FUNCTION_BLOCK PhysicsRulesWorkPieces (* Basic Function Block Type *)
  (* Standard: 61499-2 *)
  (* Version 0.0, 6/8/2016, Andrei, nxtControl GmbH, Template *)
  PACKAGE Main;
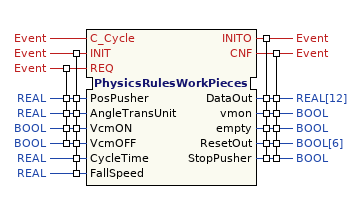
  EVENT_INPUT
    C_Cycle;
    INIT WITH PosPusher, AngleTransUnit, VcmON, VcmOFF, CycleTime, FallSpeed;
    REQ WITH PosPusher, AngleTransUnit, VcmON, VcmOFF; (* Normal Execution Request *)
  END_EVENT
  EVENT_OUTPUT
    INITO WITH DataOut, vmon, empty, ResetOut, StopPusher;
    CNF WITH DataOut, vmon, empty, ResetOut, StopPusher; (* Execution Confirmation *)
  END_EVENT
  VAR_INPUT
    PosPusher : REAL;
    AngleTransUnit : REAL;
    VcmON : BOOL;
    VcmOFF : BOOL;
    CycleTime : REAL;
    FallSpeed : REAL;
  END_VAR
  VAR_OUTPUT
    DataOut : ARRAY [0..11] OF REAL;
    vmon : BOOL;
    empty : BOOL;
    ResetOut : ARRAY [0..5] OF BOOL;
    StopPusher : BOOL;
  END_VAR
  VAR
    b : INT := 0;
    bo : INT := 0;
    bc : INT;
    bt : INT := 4; (* Number of balls *)
    Xe : ARRAY [0..3] OF REAL;
    Reset : ARRAY [0..5] OF BOOL;
    Data : ARRAY [0..11] OF REAL;
    Attached : ARRAY [0..5] OF BOOL;
    PusherStopped : BOOL;
    TUstopLeft : BOOL;
    TUstopRight : BOOL;
    MgzEmpty : BOOL := TRUE;
  END_VAR
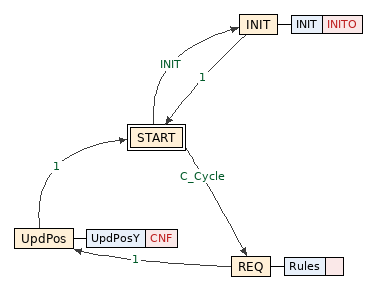
  EC_STATES
    START; (* Initial State *)
    REQ : Rules; (* Normal execution *)
    INIT : INIT -> INITO;
    UpdPos : UpdPosY -> CNF;
  END_STATES
  EC_TRANSITIONS
    REQ TO UpdPos := 1;
    START TO INIT := INIT;
    INIT TO START := 1;
    START TO REQ := C_Cycle;
    UpdPos TO START := 1;
  END_TRANSITIONS
  ALGORITHM Rules IN ST: (* Normally executed algorithm *)
// Check for conflicts.

FOR b:=0 TO 11 BY 2 DO
	// In y axis.
	// Conditions to enter falling state.
	// First entering the model. If the piston is retracted.
	IF (Data[b+1]<236.0) AND (Data[b]<277.0) THEN
		Reset[b/2] := FALSE;
	END_IF;

	//Dropped in incorrect position.
	IF (Data[b+1]<269.0) AND (Data[b] > 278.0) AND (Data[b]<610) THEN
		Reset[b/2] := FALSE;
	END_IF;

	// Conditions to stop vertical movement.
	// If another workpiece is under the present workpiece, stop vertical mov, except IF it was incorrectly placed.
	FOR bc:=0 TO 11 BY 2 DO
		IF (bc < b) AND (Data[b+1]+30.0 > Data[bc+1]) AND (Data[b]+60>Data[bc]) AND (Data[b]-60.0<Data[bc])
		AND (Data[bc+1]<240.0) THEN
			Reset[b/2] := TRUE;
		END_IF;
	END_FOR;
	// If pusher is under the workpiece, stop workpiece.
	IF (Data[b+1]<236.0) AND (Data[b+1]>=205.0)	AND (115.0+PosPusher > 6.0) AND (Data[b]<168.1) THEN
		Reset[b/2] := TRUE;
	END_IF;
	// Stop pusher IF a wp is falling in front OF it.
	IF (Data[b+1]<235.0) AND (Data[b+1]>208.0) AND (115.0+PosPusher > 6.0) AND (Data[b]<168.1) THEN
		PusherStopped := TRUE;
	END_IF;
	// Reached bottom OF buffer.
	IF (Data[b+1] > 236.0) AND ((Data[b]<=277.0) OR (Data[b]>=610.0)) THEN
		Data[b+1] := 236.0;
		Reset[b/2] := TRUE;
	END_IF;
	// Piece dropped Attached wrong position
	IF (Data[b+1] > 269.0) AND (Data[b]>278.0) AND (Data[b]<610.0) THEN
		Data[b+1] := 277.0;
		Reset[b/2] := TRUE;
	END_IF;

	// In x axis.
	// Getting pushed by the piston.
	IF (Data[b+1] > 235.9) AND (Data[b+1] < 236.1) AND (115.0+PosPusher+162.0 > Data[b]) AND
		(b < 2) THEN
		Data[b] := 115.0+PosPusher+162.0;
	END_IF;

	IF (Data[b+1] > 235.9) AND (Data[b+1] < 236.1) AND (115.0+PosPusher+162.0 > Data[b])
	AND (b>=2) AND NOT(Data[b]>214 AND (Data[b-2]<337) AND (Data[b-2]>276) AND Data[b-1]>205.9 AND Data[b-1]<236.1)  THEN
		Data[b] := 115.0+PosPusher+162.0;
	END_IF;

	// StopPusher cylinder IF two pieces are IN front OF it.
	IF (b>=2) AND (Data[b]>214 AND (Data[b-2]<337) AND (Data[b-2]>276) AND Data[b-1]>205.9 AND Data[b-1]<236.1) AND (PosPusher>=-57) THEN
		PusherStopped := TRUE;
	END_IF;

	// Getting pushed by previous workpiece in front of the pusher only.
	IF (b>=2) AND (Data[b+1]>235.9) AND (Data[b+1]<236.1) AND (Data[b]+60>Data[b-2]) AND (Data[b]<277.0) AND (Data[b-1]<236.1)
	AND NOT(Attached[(b-2)/2]) THEN
		Data[b-2] := Data[b]+60.0;
	END_IF;

	// Getting moved BY transfer unit.
	IF (Data[b]>=260.0) AND (Data[b]<=278) AND (AngleTransUnit>=179.9) AND (VcmON) AND NOT(VcmOFF) THEN
		Attached[b/2] := TRUE;
	ELSIF VcmOFF THEN
		Attached[b/2] := FALSE;
	END_IF;

	IF Attached[b/2] THEN
		Data[b] := 477.0 + (COS(AngleTransUnit*3.14159265/180.0))*170.0 - 30;
		Data[b+1] := 236.0 - (SIN(AngleTransUnit*3.14159265/180.0))*170.0;
	END_IF;

	// Mgz sensor.
	IF (Data[b] <= 198) AND (Data[b+1]>222) AND (Data[b+1]<237) THEN
		MgzEmpty := FALSE;
	END_IF;
END_FOR;

IF PusherStopped THEN
	StopPusher := TRUE;
	PusherStopped := FALSE;
ELSE
	StopPusher := FALSE;
END_IF;

// Sensors
IF Attached[0] OR Attached[1] OR Attached[2] OR Attached[3] OR Attached[4] OR Attached[5] THEN
	vmon := TRUE;
ELSE
	vmon := FALSE;
END_IF;

IF (PosPusher>-80) OR NOT(MgzEmpty) THEN
	empty := FALSE;
	MgzEmpty := TRUE;
ELSE
	empty := TRUE;
END_IF;
  END_ALGORITHM
  ALGORITHM INIT IN ST:
Data[0] := 168;
Data[1] := 206;
Data[2] := 168;
Data[3] := 175;
Data[4] := 168;
Data[5] := 144;
Data[6] := 168;
Data[7] := 113;
Data[8] := 168;
Data[9] := 82;
Data[10] := 168;
Data[11] := 51;
DataOut := Data;
  END_ALGORITHM
  ALGORITHM UpdPosY IN ST:
ResetOut := Reset;

FOR b := 0 TO 5 BY 1 DO
	IF NOT(Reset[b]) THEN
		Data[(b*2+1)] := Data[(b*2+1)] + FallSpeed*CycleTime;
	END_IF;

	// MOVE TO RIGHT once correct position is reached.
	IF (Data[b*2]>610) AND (Data[b*2+1]>235.9) AND (Data[b*2]<1000) AND NOT(Attached[b]) THEN
		Data[b*2] := Data[b*2] + FallSpeed*2*CycleTime;
	END_IF;
END_FOR;

DataOut := Data;
  END_ALGORITHM
END_FUNCTION_BLOCK
